PROGRAM MAIN

VAR

	EKE: BOOL; 
	STEP: INT :=1;
	
	TMR100: TON;
	stage: INT :=0;
	IC_CASE: INT :=0;
	
	START_STR: F_TRIG;
	START_G6: R_TRIG;
	I_RS4_PICKING_DONE: BOOL;
	START_STRAIGHTENER: R_TRIG;
	READY_1: BOOL;
	READY_2: BOOL;
	RR: BOOL;
	RX: R_TRIG;
	TRIG_IND2: R_TRIG;
END_VAR


//INPUT_CARTESSIAN(); 
INPUT_G6();
INDEXING();
INDEXING_2();
INPUT_PROG();
LOADER_RS4();
SORTER_RS4();
STRAIGHTENING_PROG_1();

(*
//EXECUTE_FUNCTION(INPUT_VAR.I_FUNCTION_NAME);

//LOAD_FUKUDA();
//MOVE STATION & JIG INDEX 


(************.::INDEXING 1 OPERATION::.***********) 
//LOADER_RS4_VAR.I_LOADER_RS4_READY_TAKEUP AND INPUT_G6_VAR.I_G6_READY_PLACING 
(*
IF INPUT_G6_VAR.I_G6_START_TAKEUP  THEN
	READY_1 :=TRUE;	
END_IF
IF LOADER_RS4_VAR.I_LOADER_RS4_START_PLACING  THEN
	READY_2 :=TRUE;
END_IF
*)

//START ROTATION INDEXING 1
READY_1 :=INPUT_G6_VAR.I_G6_START_TAKEUP;
READY_2 :=LOADER_RS4_VAR.I_LOADER_RS4_START_PLACING;
IF INDEXING_1_VAR.READY_STRAIGTHEN THEN
	READY_1 :=FALSE;	
	READY_2 :=FALSE;	
END_IF

IF READY_1 AND READY_2 AND INDEXING_1_VAR.I_INDEXING_1_ROTATION_DONE THEN//READY_PLACING THEN
	RR:=TRUE;
	RX(CLK:=RR);
	INDEXING_1_VAR.O_ROTATION_START:=RX.Q;
ELSE
	RR:=FALSE;
//RX(IN:=FALSE);
	RX(CLK:=FALSE);
END_IF


//START ROTATION INDEXING 2
IF SORTER_RS4_VAR.I_SORTER_RS4_END_CARRIER AND LOADER_RS4_VAR.I_LOADER_RS4_END_CARRIER THEN
	TRIG_IND2(CLK:=TRUE);
	INDEXING_2_VAR.O_ROTATION_START:=TRIG_IND2.Q;
	SORTER_RS4_VAR.I_SORTER_RS4_END_CARRIER:=FALSE;
	LOADER_RS4_VAR.I_LOADER_RS4_END_CARRIER:=FALSE;
	ELSE
	TRIG_IND2(CLK:=FALSE);
END_IF
*)
//CARTESSIAN INPUT
IF FLAG_VAR.ALLOW_EXECUTE_LOAD_FUKUDA THEN 
	IF INPUT_VAR.I_CASE=100 THEN
		INPUT_VAR.I_CASE:=0;
		IC_CASE:=0;	
		END_IF			
	LOAD_FUKUDA();
END_IF
IF FLAG_VAR.ALLOW_EXECUTE_RETURN_FUKUDA THEN 
	IF INPUT_VAR.I_CASE=100 THEN
		INPUT_VAR.I_CASE:=0;
		IC_CASE:=0;
	END_IF	
	RETURN_FUKUDA();	
END_IF

IF FLAG_VAR.ALLOW_EXECUTE_LOAD_LASER THEN 
	IF SORTER_VAR.I_CASE=100 THEN
		SORTER_VAR.I_CASE:=0;
		IC_CASE:=0;	
		END_IF			 
	LOAD_LASER();
END_IF
IF FLAG_VAR.ALLOW_EXECUTE_RETURN_LASER THEN 
	IF SORTER_VAR.I_CASE=100 THEN
		SORTER_VAR.I_CASE:=0;
		IC_CASE:=0;
	END_IF	
	RETURN_LASER();	
END_IF

IF FLAG_VAR.ALLOW_EXECUTE_LOAD_NG THEN 
	LOAD_NG();	
END_IF

IF FLAG_VAR.ALLOW_EXECUTE_RETURN_NG THEN 
	RETURN_NG();	
END_IF

END_PROGRAM

(* stored: Version 1.1.0.1, ProductVersion 3.1.4020.12
   POU MAIN: Id {7c8980ea-33fa-43d8-a78f-e548a5c87807}, SpecialFunc None *)
